(* IEC 61131-3 sources: julia_exos_development/test/suite/template_generation/expected/ros_topics_typ_cpp_napi/ros_topics, 2 files *)

(* ---- ros_topics_typ.typ ---- *)
TYPE
	ros_topic_point_typ : 	STRUCT  (*this expresses velocity in free space broken into its linear and angular parts.*)
		y : LREAL;
		z : LREAL;
		x : LREAL;
	END_STRUCT;
	ros_topic_vector3_typ : 	STRUCT  (*this expresses velocity in free space broken into its linear and angular parts.*)
		y : LREAL;
		z : LREAL;
		x : LREAL;
	END_STRUCT;
	ros_topic_twist_typ : 	STRUCT  (*This expresses velocity in free space broken into its linear and angular parts.*)
		angular : ros_topic_vector3_typ; (*SUB*)
		linear : ros_topic_vector3_typ; (*SUB*)
	END_STRUCT;
	ros_topic_twistCor_typ : 	STRUCT  (*This expresses velocity in free space with uncertainty.*)
		twist : ros_topic_twist_typ;
		covariance : ARRAY[0..63]OF LREAL; (*Row-major representation of the 6x6 covariance matrix
The orientation parameters use a fixed-axis representation. In order, the parameters are:
 (x, y, z, rotation about X axis, rotation about Y axis, rotation about Z axis)*)
	END_STRUCT;
	ros_topic_quaternion_typ : 	STRUCT  (*This represents an orientation in free space in quaternion form.*)
		y : LREAL;
		z : LREAL;
		w : LREAL;
		x : LREAL;
	END_STRUCT;
	ros_topic_odemety_point_typ : 	STRUCT  (*This contains the position of a point in free space*)
		y : LREAL;
		z : LREAL;
		x : LREAL;
	END_STRUCT;
	ros_topic_pose_typ : 	STRUCT  (*A representation of pose in free space, composed of position and orientation. *)
		position : ros_topic_point_typ;
		orientation : ros_topic_quaternion_typ;
	END_STRUCT;
	ros_topic_poseCor_typ : 	STRUCT  (*This represents a pose in free space with uncertainty.*)
		pose : ros_topic_pose_typ;
		covariance : ARRAY[0..63]OF LREAL; (*Row-major representation of the 6x6 covariance matrix
The orientation parameters use a fixed-axis representation. In order, the parameters are:
 (x, y, z, rotation about X axis, rotation about Y axis, rotation about Z axis)*)
	END_STRUCT;
	ros_topic_time_typ : 	STRUCT
		nsec : UDINT;
		sec : UDINT;
	END_STRUCT;
	ros_topic_header_typ : 	STRUCT
		stamp : ros_topic_time_typ;
		seq : UDINT;
		frame_id : STRING[20];
	END_STRUCT;
	ros_topic_odemety_typ : 	STRUCT
		pose : ros_topic_poseCor_typ; (*PUB*)
		twist : ros_topic_twistCor_typ; (*PUB*)
		header : ros_topic_header_typ; (*PUB*)
	END_STRUCT;
	ros_config_typ : 	STRUCT
		maxSpeed : LREAL := 2; (*SUB*)
		minSpeed : LREAL := -2; (*SUB*)
		baseWidth : LREAL := 0.53; (*SUB*)
	END_STRUCT;
	ros_topics_typ : 	STRUCT
		odemetry : ros_topic_odemety_typ; (*PUB*)
		twist : ros_topic_twist_typ; (*SUB*)
		config : ros_config_typ; (*SUB*)
	END_STRUCT;
END_TYPE

(* ---- ros_topics.fun ---- *)
FUNCTION_BLOCK ros_topics_typInit
    VAR_OUTPUT
        Handle : UDINT;
    END_VAR
END_FUNCTION_BLOCK

FUNCTION_BLOCK ros_topics_typCyclic
    VAR_INPUT
        Enable : BOOL;
        Start : BOOL;
        Handle : UDINT;
        pros_topics_typ : REFERENCE TO ros_topics_typ;
    END_VAR
    VAR_OUTPUT
        Connected : BOOL;
        Operational : BOOL;
        Error : BOOL;
    END_VAR
    VAR
        _Start : BOOL;
        _Enable : BOOL;
    END_VAR
END_FUNCTION_BLOCK

FUNCTION_BLOCK ros_topics_typExit
    VAR_INPUT
        Handle : UDINT;
    END_VAR
END_FUNCTION_BLOCK
